TYPE CurrentStep :
STRUCT
	number : INT;
	actionNumber : INT;
	elapsedTime : TIME;
//	entryAction : BOOL := TRUE;
//	exitAction : BOOL;
//	entryDone : BOOL;
//	exitDone : BOOL;
	
	actionDone : BOOL;
END_STRUCT
END_TYPE

(* stored: Version 1.1.0.1, ProductVersion 3.1.4024.11
   DUT CurrentStep: Id {c55e124c-9bca-4328-84c4-ddf821e192e2} *)
